FUNCTION_BLOCK FB_Load
VAR
	nCount							: INT;
END_VAR

// =========================================================
(* Product parameters *)
(* Product parameter - Set load on true *)
IF (stTempLoad.stTempCmd.bLoadPparams AND NOT stTempLoad.stTempState.bPparamLoad) THEN
	stTempLoad.stTempCmd.bLoadPparams:=
	stTempLoad.stTempState.bPparamLoaded:= FALSE;
	stTempLoad.stTempState.bPparamLoad:= TRUE;
	FOR nCount:=cnPfwTempCtrlFirst TO cnPfwTempCtrlLast DO
		aaaPfwTempPparamFromHmi[nCount].bLoadParams:= TRUE;
	END_FOR
END_IF
(* Product parameter - check load is done *)
IF stTempLoad.stTempState.bPparamLoad THEN
	stTempLoad.stTempState.bPparamLoad:= FALSE;
	FOR nCount:=cnPfwTempCtrlFirst TO cnPfwTempCtrlLast DO
		IF aaaPfwTempPparamFromHmi[nCount].bLoadParams THEN
			stTempLoad.stTempState.bPparamLoad:= TRUE;
		END_IF
	END_FOR
	stTempLoad.stTempState.bPparamLoaded:= NOT stTempLoad.stTempState.bPparamLoad;
END_IF

(* Machine parameters *)
(* Machine parameter - Set load on true *)
IF (stTempLoad.stTempCmd.bLoadMparams AND NOT stTempLoad.stTempState.bMparamLoad) THEN
	stTempLoad.stTempCmd.bLoadMparams:=
	stTempLoad.stTempState.bMparamLoaded:= FALSE;
	stTempLoad.stTempState.bMparamLoad:= TRUE;
	FOR nCount:=cnPfwTempCtrlFirst TO cnPfwTempCtrlLast DO
		aaaPfwTempMparamFromHmi[nCount].bLoadParams:= TRUE;
	END_FOR
END_IF
(* Machine parameter - check load is done *)
IF stTempLoad.stTempState.bMparamLoad THEN
	stTempLoad.stTempState.bMparamLoad:= FALSE;
	FOR nCount:=cnPfwTempCtrlFirst TO cnPfwTempCtrlLast DO
		IF aaaPfwTempMparamFromHmi[nCount].bLoadParams THEN
			stTempLoad.stTempState.bPparamLoad:= TRUE;
		END_IF
	END_FOR
	stTempLoad.stTempState.bMparamLoaded:= NOT stTempLoad.stTempState.bMparamLoad;
END_IF


(* Supply lines *)
(* Supply lines - Set load on true *)
IF (stTempLoad.stTempCmd.bLoadSupplyParams AND NOT stTempLoad.stTempState.bSupplyParamsLoad) THEN
	stTempLoad.stTempCmd.bLoadSupplyParams:=
	stTempLoad.stTempState.bSupplyParamsLoaded:= FALSE;
	stTempLoad.stTempState.bSupplyParamsLoad:= TRUE;
	FOR nCount:=cnPfwAppSupplyFirst TO cnPfwAppSupplyLast DO
		stPfwSupplyLineCfg[nCount].bLoadParams:= TRUE;
	END_FOR
END_IF
(* Supply lines - check load is done *)
IF stTempLoad.stTempState.bSupplyParamsLoad THEN
	stTempLoad.stTempState.bSupplyParamsLoad:= FALSE;
	FOR nCount:=cnPfwAppSupplyFirst TO cnPfwAppSupplyLast DO
		IF stPfwSupplyLineCfg[nCount].bLoadParams THEN
			stTempLoad.stTempState.bSupplyParamsLoad:= TRUE;
		END_IF
	END_FOR
	stTempLoad.stTempState.bSupplyParamsLoaded:= NOT stTempLoad.stTempState.bSupplyParamsLoad;
END_IF
// =========================================================

END_FUNCTION_BLOCK

(* stored: Version 1.1.0.1
   POU FB_Load: Id {508d3fb0-e11d-4506-9cb5-c1b7bfcf7ffc}, SpecialFunc None *)
